{attribute 'qualified_only'}
{attribute 'strict'}
TYPE E_Trolley :
(
	enum_member := 0
);
END_TYPE

(* stored: Version 1.1.0.1, ProductVersion 3.1.4024.12
   DUT E_Trolley: Id {631bd5bc-a8eb-467e-922f-2faa5112a34b} *)
